(* PLC project Unnamed, Unknown Unnamed 1 *)
(* stored: creationDateTime 2026-09-24T12:23:45, modificationDateTime 2026-09-24T14:53:47 *)

PROGRAM TankFill
  VAR
    TankFillAuto_Cmd : BOOL;  (* Internal automatic fill latch/command *)
    TankValveOpen : BOOL;  (* Discrete command/status for the fill valve *)
    Estop_Cmd : BOOL;  (* Emergency-stop input; TRUE forces automatic fill to stop *)
    TankLevelHi_Alarm : BOOL;  (* High-level alarm state *)
    TankLevelLo_Alarm : BOOL;  (* Low-level alarm state *)
    TankLevel_LIT : REAL;  (* Measured tank level in feet *)
    TankEmpty_SP : REAL := 2.0;  (* Automatic fill start setpoint (2.0 ft) *)
    TankFull_SP : REAL := 8.0;  (* Automatic fill stop setpoint (8.0 ft) *)
    TankLoAlarm_SP : REAL := 1.0;  (* Low-level alarm setpoint (1.0 ft) *)
    TankHiAlarm_SP : REAL := 9.0;
  END_VAR

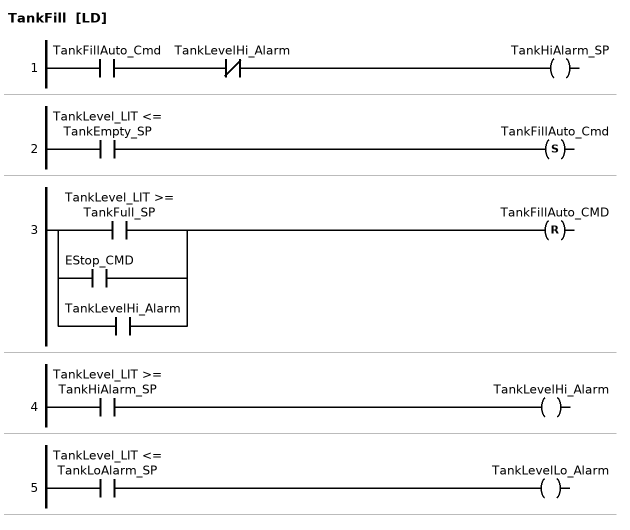
(* LD diagram, written out as Structured Text *)
TankHiAlarm_SP := TankFillAuto_Cmd AND NOT TankLevelHi_Alarm;
IF TankLevel_LIT <= TankEmpty_SP THEN TankFillAuto_Cmd := TRUE; END_IF;
IF (TankLevel_LIT >= TankFull_SP) OR EStop_CMD OR TankLevelHi_Alarm THEN TankFillAuto_CMD := FALSE; END_IF;
TankLevelHi_Alarm := TankLevel_LIT >= TankHiAlarm_SP;
TankLevelLo_Alarm := TankLevel_LIT <= TankLoAlarm_SP;
END_PROGRAM

CONFIGURATION Config0
  RESOURCE Res0 ON PLC
    TASK task0(INTERVAL := T#20ms, PRIORITY := 0);
    PROGRAM instance0 WITH task0 : TankFill;
  END_RESOURCE
END_CONFIGURATION
